// TIA Portal project "babu_3WayTrafficComparators" (V15)

(* hardware
DEVICE "S7-1200 station_1"  S7-1200 Station
   slot 0: "Rack_0"  S7-1200 Rack  Rack  V1.0
   slot 1: "PLC_1"  CPU 1212C DC/DC/DC  6ES7 212-1AE40-0XB0  V4.2
*)

// ===== PLC "PLC_1"  CPU 1212C DC/DC/DC =====

VAR_GLOBAL   // PLC tag table "Default tag table"
   "PUSH BUTTON" AT %M0.0 : Bool;
   "PB MEMORY" AT %M0.1 : Bool;
   "INITIALIZE" AT %M0.2 : Bool;
   "INITIALIZE ALL LIGHTS" AT %M0.3 : Bool;
   "START" AT %M0.4 : Bool;
   "START 30" AT %M0.5 : Bool;
   "START 10" AT %M0.6 : Bool;
   "R1" AT %Q0.0 : Bool;
   "R2" AT %Q0.1 : Bool;
   "G3" AT %Q0.2 : Bool;
   "Y1" AT %Q0.3 : Bool;
   "G1" AT %Q0.4 : Bool;
   "R3" AT %Q0.5 : Bool;
   "Y2" AT %Q0.6 : Bool;
   "G2" AT %Q0.7 : Bool;
   "Y3" AT %Q1.0 : Bool;
   "RESET TIMER" AT %M0.7 : Bool;
END_VAR

// folder: System blocks/Program resources

DATA_BLOCK "IEC_Timer_0_DB_2"   // DB4
{ S7_Optimized_Access := 'TRUE' }
AUTHOR : Simatic
FAMILY : IEC
NAME : IEC_TMR
VERSION : 1.0
// stored: InstanceOfName IEC_TIMER
"IEC_TIMER"
BEGIN
END_DATA_BLOCK

DATA_BLOCK "IEC_Timer_0_DB_3"   // DB5
{ S7_Optimized_Access := 'TRUE' }
AUTHOR : Simatic
FAMILY : IEC
NAME : IEC_TMR
VERSION : 1.0
// stored: InstanceOfName IEC_TIMER
"IEC_TIMER"
BEGIN
END_DATA_BLOCK

// folder: (top level)

ORGANIZATION_BLOCK "Main"   // OB1, LAD, ProgramCycle
TITLE = "Main Program Sweep (Cycle)"
{ S7_Optimized_Access := 'TRUE' }
VERSION : 0.1
   VAR_INPUT
      Initial_Call : Bool;   // Initial call of this OB
      Remanence : Bool;   // =True, if remanent data are available
   END_VAR
BEGIN

REGION Network 1: INITIALIZE
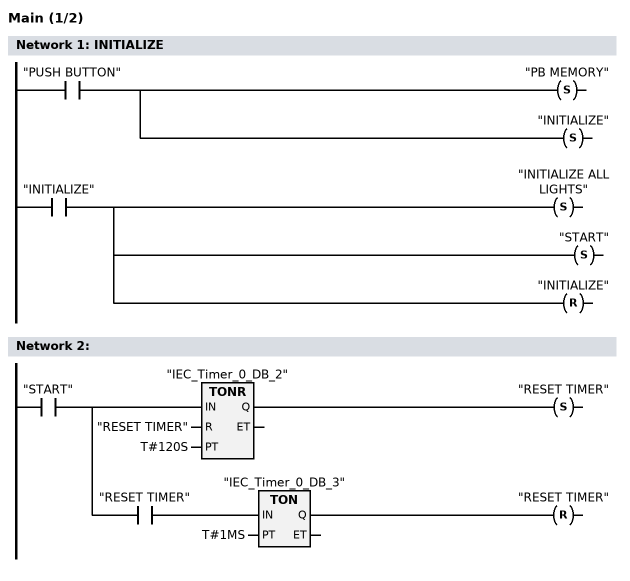
   RUNG wire#powerrail
      Contact( "PUSH BUTTON" )
      wire#w1
      S_Coil( "PB MEMORY" )
   END_RUNG
   RUNG wire#w1
      S_Coil( "INITIALIZE" )
   END_RUNG
   RUNG wire#powerrail
      Contact( "INITIALIZE" )
      wire#w2
      S_Coil( "INITIALIZE ALL LIGHTS" )
   END_RUNG
   RUNG wire#w2
      S_Coil( "START" )
   END_RUNG
   RUNG wire#w2
      R_Coil( "INITIALIZE" )
   END_RUNG
   // the same network as SCL:
   IF "PUSH BUTTON" THEN
       "PB MEMORY" := TRUE;
       "INITIALIZE" := TRUE;
   END_IF;
   IF "INITIALIZE" THEN
       "INITIALIZE ALL LIGHTS" := TRUE;
       "START" := TRUE;
       "INITIALIZE" := FALSE;
   END_IF;
END_REGION

REGION Network 2
   "IEC_Timer_0_DB_2".TONR(IN := "START", R := "RESET TIMER", PT := T#120S);
   IF "IEC_Timer_0_DB_2".Q THEN "RESET TIMER" := TRUE; END_IF;
   "IEC_Timer_0_DB_3".TON(IN := "START" AND "RESET TIMER", PT := T#1MS);
   IF "IEC_Timer_0_DB_3".Q THEN "RESET TIMER" := FALSE; END_IF;
END_REGION

REGION Network 3
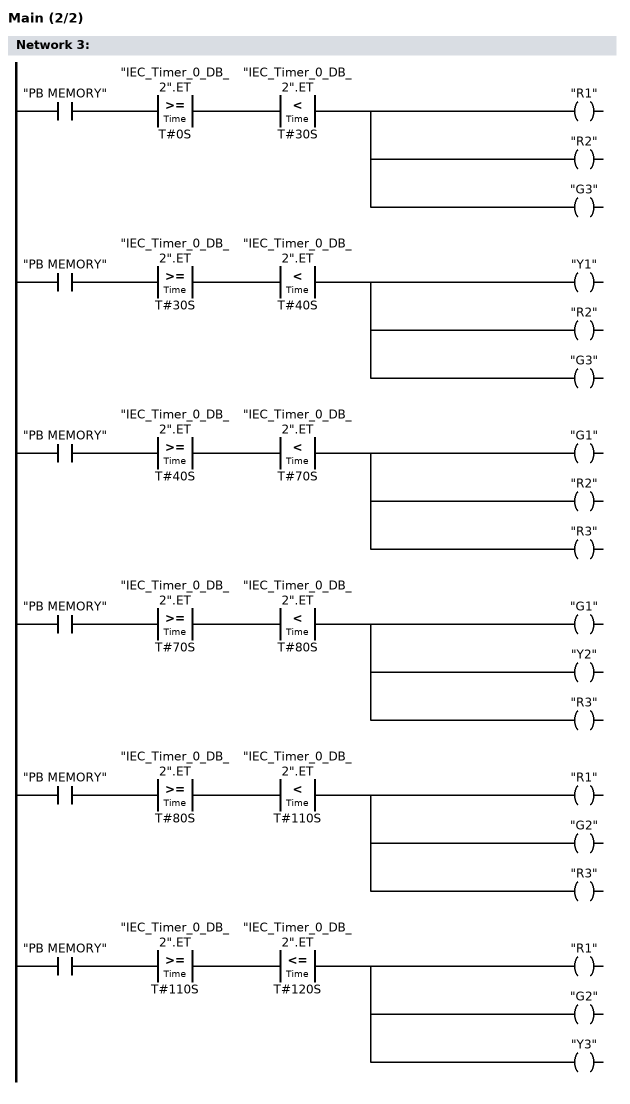
   RUNG wire#powerrail
      Contact( "PB MEMORY" )
      { S7_Templates := "SrcType := Time" } GE_Contact(in1 := "IEC_Timer_0_DB_2".ET, in2 := T#0S)
      { S7_Templates := "SrcType := Time" } LT_Contact(in1 := "IEC_Timer_0_DB_2".ET, in2 := T#30S)
      wire#w1
      Coil( "R1" )
   END_RUNG
   RUNG wire#w1
      Coil( "R2" )
   END_RUNG
   RUNG wire#w1
      Coil( "G3" )
   END_RUNG
   RUNG wire#powerrail
      Contact( "PB MEMORY" )
      { S7_Templates := "SrcType := Time" } GE_Contact(in1 := "IEC_Timer_0_DB_2".ET, in2 := T#30S)
      { S7_Templates := "SrcType := Time" } LT_Contact(in1 := "IEC_Timer_0_DB_2".ET, in2 := T#40S)
      wire#w2
      Coil( "Y1" )
   END_RUNG
   RUNG wire#w2
      Coil( "R2" )
   END_RUNG
   RUNG wire#w2
      Coil( "G3" )
   END_RUNG
   RUNG wire#powerrail
      Contact( "PB MEMORY" )
      { S7_Templates := "SrcType := Time" } GE_Contact(in1 := "IEC_Timer_0_DB_2".ET, in2 := T#40S)
      { S7_Templates := "SrcType := Time" } LT_Contact(in1 := "IEC_Timer_0_DB_2".ET, in2 := T#70S)
      wire#w3
      Coil( "G1" )
   END_RUNG
   RUNG wire#w3
      Coil( "R2" )
   END_RUNG
   RUNG wire#w3
      Coil( "R3" )
   END_RUNG
   RUNG wire#powerrail
      Contact( "PB MEMORY" )
      { S7_Templates := "SrcType := Time" } GE_Contact(in1 := "IEC_Timer_0_DB_2".ET, in2 := T#70S)
      { S7_Templates := "SrcType := Time" } LT_Contact(in1 := "IEC_Timer_0_DB_2".ET, in2 := T#80S)
      wire#w4
      Coil( "G1" )
   END_RUNG
   RUNG wire#w4
      Coil( "Y2" )
   END_RUNG
   RUNG wire#w4
      Coil( "R3" )
   END_RUNG
   RUNG wire#powerrail
      Contact( "PB MEMORY" )
      { S7_Templates := "SrcType := Time" } GE_Contact(in1 := "IEC_Timer_0_DB_2".ET, in2 := T#80S)
      { S7_Templates := "SrcType := Time" } LT_Contact(in1 := "IEC_Timer_0_DB_2".ET, in2 := T#110S)
      wire#w5
      Coil( "R1" )
   END_RUNG
   RUNG wire#w5
      Coil( "G2" )
   END_RUNG
   RUNG wire#w5
      Coil( "R3" )
   END_RUNG
   RUNG wire#powerrail
      Contact( "PB MEMORY" )
      { S7_Templates := "SrcType := Time" } GE_Contact(in1 := "IEC_Timer_0_DB_2".ET, in2 := T#110S)
      { S7_Templates := "SrcType := Time" } LE_Contact(in1 := "IEC_Timer_0_DB_2".ET, in2 := T#120S)
      wire#w6
      Coil( "R1" )
   END_RUNG
   RUNG wire#w6
      Coil( "G2" )
   END_RUNG
   RUNG wire#w6
      Coil( "Y3" )
   END_RUNG
   // the same network as SCL:
   "R1" := "PB MEMORY" AND ("IEC_Timer_0_DB_2".ET >= T#0S) AND ("IEC_Timer_0_DB_2".ET < T#30S);
   "R2" := "R1";
   "G3" := "R1";
   "Y1" := "PB MEMORY" AND ("IEC_Timer_0_DB_2".ET >= T#30S) AND ("IEC_Timer_0_DB_2".ET < T#40S);
   "R2" := "Y1";
   "G3" := "Y1";
   "G1" := "PB MEMORY" AND ("IEC_Timer_0_DB_2".ET >= T#40S) AND ("IEC_Timer_0_DB_2".ET < T#70S);
   "R2" := "G1";
   "R3" := "G1";
   "G1" := "PB MEMORY" AND ("IEC_Timer_0_DB_2".ET >= T#70S) AND ("IEC_Timer_0_DB_2".ET < T#80S);
   "Y2" := "G1";
   "R3" := "G1";
   "R1" := "PB MEMORY" AND ("IEC_Timer_0_DB_2".ET >= T#80S) AND ("IEC_Timer_0_DB_2".ET < T#110S);
   "G2" := "R1";
   "R3" := "R1";
   "R1" := "PB MEMORY" AND ("IEC_Timer_0_DB_2".ET >= T#110S) AND ("IEC_Timer_0_DB_2".ET <= T#120S);
   "G2" := "R1";
   "Y3" := "R1";
END_REGION
END_ORGANIZATION_BLOCK